FUNCTION_BLOCK Test_TStreamAdd_Read_DINT EXTENDS T_UnitTestBase
VAR
    Stream  : T_Stream(StreamLength := 2);
    ArgType : E_ArgTypeId := E_ArgTypeId.Type_DINT;
END_VAR

{attribute 'analysis' := '-33'} // inhibit unused variable warning
METHOD RunTest
Stream.Init(2);

// add a DINT...
Stream.SetNextArgTypeId(ArgType);
Stream.Add_DINT(12345678);

Stream.SetReadPosition(0);

// check next arg type is correct...
AssertEquals_INT(Expected     := ArgType,
                           Actual       := Stream.GetNextArgTypeId(),
                           Message := 'Stream.GetNextArgTypeId()');

// check next value...	
AssertEquals_DINT(Expected     := 12345678,
                            Actual       := Stream.Read_DINT(),
                            Message := 'Stream.Read_DINT()');

// check we are at the end of the stream..							
AssertEquals_UDINT(Expected     := Stream.StreamLength,
                             Actual       := Stream.ReadPosition,
                             Message := 'Stream.ReadPosition');

TestCompleted := TRUE;
END_METHOD

END_FUNCTION_BLOCK

(* stored: Version 1.1.0.1, ProductVersion 3.1.4024.12
   POU Test_TStreamAdd_Read_DINT: Id {0dd6c6a4-a29e-4502-8f8a-33d512d8e3b5}, SpecialFunc None
   Method RunTest: Id {81104695-2ca0-4a2d-9b7d-cf4929d020f8} *)
